// TIA Portal V21 export
TYPE "Std_eResponseReadMalfunctionList"
   STRUCT
      idle { ExternalVisible := 'False'} : Int := 0;
      setting_valve_to_inactive { ExternalVisible := 'False'} : Int := 1;
      getting_malfunction_count { ExternalVisible := 'False'} : Int := 2;
      transferring { ExternalVisible := 'False'} : Int := 3;
      done { ExternalVisible := 'False'} : Int := 4;
      no_entries_in_malfunction_list { ExternalVisible := 'False'} : Int := 5;
      error_while_transmitting_data_to_vtem { ExternalVisible := 'False'} : Int := 6;
      aborting { ExternalVisible := 'False'} : Int := 7;
      resetting { ExternalVisible := 'False'} : Int := 8;
      FB_needs_rising_edge_xExecute { ExternalVisible := 'False'} : Int := 10;
      reserved { ExternalVisible := 'False'} : Int := 100;
      invalid_SetValveMode { ExternalVisible := 'False'} : Int := 101;
      invalid_SetAppControl { ExternalVisible := 'False'} : Int := 102;
      invalid_SetAppOption { ExternalVisible := 'False'} : Int := 103;
      invalid_SetPointValue1 { ExternalVisible := 'False'} : Int := 104;
      invalid_SetPointValue2 { ExternalVisible := 'False'} : Int := 105;
      invalid_configuration { ExternalVisible := 'False'} : Int := 106;
      access_denied_WebConfig { ExternalVisible := 'False'} : Int := 110;
      access_denied_saving_parameterisation { ExternalVisible := 'False'} : Int := 111;
      no_license_for_this_MA { ExternalVisible := 'False'} : Int := 112;
      all_licenses_in_use { ExternalVisible := 'False'} : Int := 113;
      invalid_license_file { ExternalVisible := 'False'} : Int := 114;
      no_valve_detected { ExternalVisible := 'False'} : Int := 115;
      valve_self_calibration_running { ExternalVisible := 'False'} : Int := 116;
      invalid_Channel { ExternalVisible := 'False'} : Int := 201;
      invalid_TransferControl { ExternalVisible := 'False'} : Int := 202;
      invalid_iChooseOtherValve { ExternalVisible := 'False'} : Int := 203;
      invalid_Index { ExternalVisible := 'False'} : Int := 204;
      invalid_TransferValue { ExternalVisible := 'False'} : Int := 205;
      invalid_Combination { ExternalVisible := 'False'} : Int := 206;
      access_denied_DataInUse { ExternalVisible := 'False'} : Int := 207;
      no_data_empty_slot { ExternalVisible := 'False'} : Int := 208;
   END_STRUCT;
END_TYPE
